(* PLC project CoDeSys External Library Template, WAGO e!COCKPIT e!COCKPIT, author 3S - Smart Software Solutions GmbH *)
(* stored: creationDateTime 2019-10-29T12:22:40.8293431, version 3.5.5.30, modificationDateTime 2019-10-24T14:40:07.960949, organization 3S - Smart Software Solutions GmbH *)
(* Library project template with all possible element types, docu and a sample project structure *)

FUNCTION fnKomunikatDaneDodaj : STRING
  VAR_INPUT
    sAtrybut : STRING;
    sWartosc : STRING;
  END_VAR
  VAR_IN_OUT
    sDane : alSTRINGKomunikat;
  END_VAR

            IF sDane <> '' THEN
	sDane := CONCAT(sDane , ';');
END_IF
sDane := CONCAT(sDane , sAtrybut);
sDane := CONCAT(sDane , sWartosc);
          
END_FUNCTION
